KUKA KRL program: ho_st600_r1_1.src, ho_st600_r1_1.dat

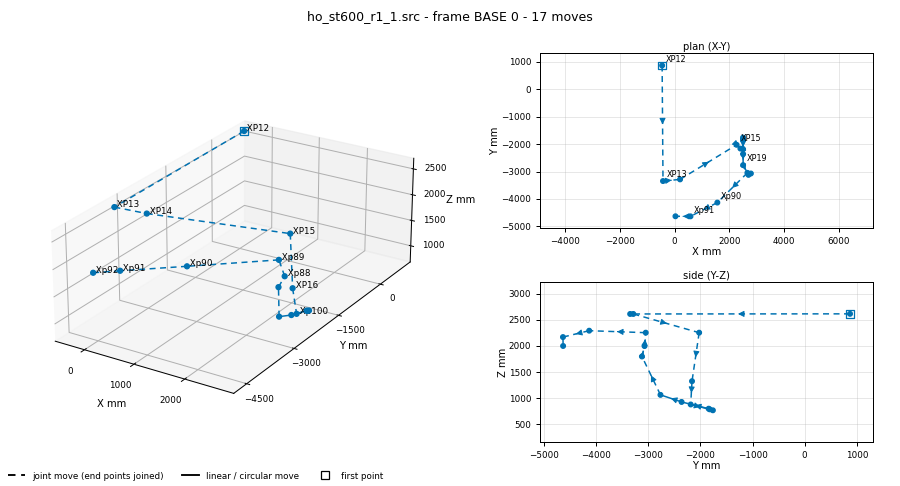
[picture p0: tool path of ho_st600_r1_1.src in frame BASE 0, 17 of 18 moves have a stored position in this frame; points joined in program order, loops and branches not executed]
--- ho_st600_r1_1.src ---
&ACCESS RVO1
&REL 93
&COMMENT Pega traseira ACTROS
&PARAM DISKPATH = KRC:\R1\Program
DEF HO_ST600_R1_1( )
;FOLD INI
  ;FOLD BASISTECH INI
    GLOBAL INTERRUPT DECL 3 WHEN $STOPMESS==TRUE DO IR_STOPM ( )
    INTERRUPT ON 3
    BAS (#INITMOV,0 )
  ;ENDFOLD (BASISTECH INI)
;FOLD GRIPPERTECH INI
USER_GRP(0,DUMMY,DUMMY,GDEFAULT)
;ENDFOLD (GRIPPERTECH INI)
  ;FOLD USER INI
    ;Make your modifications here

  ;ENDFOLD (USER INI)
;ENDFOLD (INI)

; Caracterização dos meios de produção:
; Versão Atual:
; 08/06/2013 12:00 Name: P13.050-R1 CHANGES: Pega Traseira
; Actros MGS\MGSB\LTA\LTB e STB12-13

chk_w5_wechs_ok ( )              ; CHECK GRIPPER ACTROS

;FOLD PTP P12 CONT Vel=100 % PDAT11 Tool[5]:Painel Traseiro Actros Base[0];%{PE}%R 8.2.19,%MKUKATPBASIS,%CMOVE,%VPTP,%P 1:PTP, 2:P12, 3:C_DIS, 5:100, 7:PDAT11
$BWDSTART=FALSE
PDAT_ACT=PPDAT11
FDAT_ACT=FP12
BAS(#PTP_PARAMS,100)
PTP XP12 C_DIS
;ENDFOLD
;FOLD PTP P13 Vel=100 % PDAT12 Tool[5]:Painel Traseiro Actros Base[0];%{PE}%R 8.2.20,%MKUKATPBASIS,%CMOVE,%VPTP,%P 1:PTP, 2:P13, 3:, 5:100, 7:PDAT12
$BWDSTART=FALSE
PDAT_ACT=PPDAT12
FDAT_ACT=FP13
BAS(#PTP_PARAMS,100)
PTP XP13
;ENDFOLD

;FOLD OUT 3352 'R1 busca traseira' State=TRUE ;%{PE}%R 8.2.20,%MKUKATPBASIS,%COUT,%VOUTX,%P 2:3352, 3:R1 busca traseira, 5:TRUE, 6:
$OUT[3352]=TRUE
;ENDFOLD
;FOLD WAIT FOR ( IN 3352 'Aguarda lib. Buscar traseira' );%{PE}%R 8.2.20,%MKUKATPBASIS,%CEXT_WAIT_FOR,%VEXT_WAIT_FOR,%P 2:, 4:, 5:$IN, 6:3352, 7:Aguarda lib. Buscar traseira, 9:
WAIT FOR  ( $IN[3352] )
;ENDFOLD
;FOLD OUT 3352 'R1 busca traseira' State=FALSE ;%{PE}%R 8.2.20,%MKUKATPBASIS,%COUT,%VOUTX,%P 2:3352, 3:R1 busca traseira, 5:FALSE, 6:
$OUT[3352]=FALSE
;ENDFOLD

;FOLD PTP P14 CONT Vel=100 % PDAT13 Tool[5]:Painel Traseiro Actros Base[0];%{PE}%R 8.2.19,%MKUKATPBASIS,%CMOVE,%VPTP,%P 1:PTP, 2:P14, 3:C_DIS, 5:100, 7:PDAT13
$BWDSTART=FALSE
PDAT_ACT=PPDAT13
FDAT_ACT=FP14
BAS(#PTP_PARAMS,100)
PTP XP14 C_DIS
;ENDFOLD
;FOLD PTP P15 CONT Vel=100 % PDAT14 Tool[5]:Painel Traseiro Actros Base[0];%{PE}%R 8.2.19,%MKUKATPBASIS,%CMOVE,%VPTP,%P 1:PTP, 2:P15, 3:C_DIS, 5:100, 7:PDAT14
$BWDSTART=FALSE
PDAT_ACT=PPDAT14
FDAT_ACT=FP15
BAS(#PTP_PARAMS,100)
PTP XP15 C_DIS
;ENDFOLD
;FOLD PTP P16 CONT Vel=100 % PDAT15 Tool[5]:Painel Traseiro Actros Base[0];%{PE}%R 8.2.19,%MKUKATPBASIS,%CMOVE,%VPTP,%P 1:PTP, 2:P16, 3:C_DIS, 5:100, 7:PDAT15
$BWDSTART=FALSE
PDAT_ACT=PPDAT15
FDAT_ACT=FP16
BAS(#PTP_PARAMS,100)
PTP XP16 C_DIS
;ENDFOLD

;FOLD OUT 3342 'Fora area externa' State=FALSE ;%{PE}%R 8.2.20,%MKUKATPBASIS,%COUT,%VOUTX,%P 2:3342, 3:Fora area externa, 5:FALSE, 6:
$OUT[3342]=FALSE
;ENDFOLD

;FOLD SET Z2.1/2 GRP ACTROS State= GDAT2;%{PE}%R 8.2.1,%MKUKATPGRP,%CGRP,%VGRP,%P 2:1, 4:1, 5:#NO, 6:GDAT2, 8:0, 10:0
H50(GRP,1,1,GGDAT2)
;ENDFOLD
chk_w5_grp2_opn()
;FOLD SET Z3.1/2 GRP ACTROS State=OPN GDAT3;%{PE}%R 8.2.1,%MKUKATPGRP,%CGRP,%VGRP,%P 2:2, 4:1, 5:#NO, 6:GDAT3, 8:0, 10:0
H50(GRP,2,1,GGDAT3)
;ENDFOLD
chk_w5_grp3_opn()

;FOLD PTP p100 CONT Vel=100 % PDAT71 Tool[5]:Painel Traseiro Actros Base[0];%{PE}%R 8.2.20,%MKUKATPBASIS,%CMOVE,%VPTP,%P 1:PTP, 2:p100, 3:C_DIS, 5:100, 7:PDAT71
$BWDSTART=FALSE
PDAT_ACT=PPDAT71
FDAT_ACT=Fp100
BAS(#PTP_PARAMS,100)
PTP Xp100 C_DIS
;ENDFOLD
;FOLD PTP p102 CONT Vel=100 % PDAT73 Tool[5]:Painel Traseiro Actros Base[0];%{PE}%R 8.2.20,%MKUKATPBASIS,%CMOVE,%VPTP,%P 1:PTP, 2:p102, 3:C_DIS, 5:100, 7:PDAT73
$BWDSTART=FALSE
PDAT_ACT=PPDAT73
FDAT_ACT=Fp102
BAS(#PTP_PARAMS,100)
PTP Xp102 C_DIS
;ENDFOLD

;FOLD ; POSICAO DE PEGA DA PECA;%{PE}%R 8.2.20,%MKUKATPBASIS,%CCOMMENT,%VNORMAL,%P 2:POSICAO  DE  PEGA  DA  PECA
;ENDFOLD
;FOLD LIN P18 Vel=0.5 m/s CPDAT1 Tool[5]:Painel Traseiro Actros Base[0];%{PE}%R 8.2.20,%MKUKATPBASIS,%CMOVE,%VLIN,%P 1:LIN, 2:P18, 3:, 5:0.5, 7:CPDAT1
$BWDSTART=FALSE
LDAT_ACT=LCPDAT1
FDAT_ACT=FP18
BAS(#CP_PARAMS,0.5)
LIN XP18
;ENDFOLD

IF (NOT(GHOST())) THEN
;FOLD WAIT FOR ( IN 1 'Presença de peça 1 - Actros Todos' ) AND ( IN 2 'Presença de peça 2 - Actros Todos' );%{PE}%R 8.2.20,%MKUKATPBASIS,%CEXT_WAIT_FOR,%VEXT_WAIT_FOR,%P 2:, 4:, 5:$IN, 6:1, 7:Presença de peça 1 - Actros Todos, 9:AND, 10:, 12:, 13:$IN, 14:2, 15:Presença de peça 2 - Actros Todos, 17:
WAIT FOR  ( $IN[1] ) AND ( $IN[2] )
;ENDFOLD
ENDIF

;FOLD SET Z2.1/2 GRP ACTROS State=CLO GDAT1;%{PE}%R 8.2.1,%MKUKATPGRP,%CGRP,%VGRP,%P 2:1, 4:2, 5:#NO, 6:GDAT1, 8:0, 10:0
H50(GRP,1,2,GGDAT1)
;ENDFOLD
chk_w5_grp2_clo()
;FOLD SET Z3.1/2 GRP ACTROS State=CLO GDAT4;%{PE}%R 8.2.1,%MKUKATPGRP,%CGRP,%VGRP,%P 2:2, 4:2, 5:#NO, 6:GDAT4, 8:0, 10:0
H50(GRP,2,2,GGDAT4)
;ENDFOLD
chk_w5_grp3_clo()

IF (NOT(GHOST())) THEN
;FOLD SET Ventosa ACTROS State=VACUUM GDAT5;%{PE}%R 8.2.1,%MKUKATPGRP,%CGRP,%VGRP,%P 2:6, 4:1, 5:#NO, 6:GDAT5, 8:0, 10:0
H50(GRP,6,1,GGDAT5)
;ENDFOLD
;chk_w5_grp1_vac()
ENDIF

;FOLD OUT 3350 'Solicita lib sair magazine' State=TRUE ;%{PE}%R 8.2.20,%MKUKATPBASIS,%COUT,%VOUTX,%P 2:3350, 3:Solicita lib sair magazine, 5:TRUE, 6:
$OUT[3350]=TRUE
;ENDFOLD
;FOLD WAIT FOR ( IN 3349 'Aguarda lib sair magazine' );%{PE}%R 8.2.20,%MKUKATPBASIS,%CEXT_WAIT_FOR,%VEXT_WAIT_FOR,%P 2:, 4:, 5:$IN, 6:3349, 7:Aguarda lib sair magazine, 9:
WAIT FOR  ( $IN[3349] )
;ENDFOLD
;FOLD OUT 3350 'Solicita lib sair magazine' State=FALSE ;%{PE}%R 8.2.20,%MKUKATPBASIS,%COUT,%VOUTX,%P 2:3350, 3:Solicita lib sair magazine, 5:FALSE, 6:
$OUT[3350]=FALSE
;ENDFOLD
;FOLD OUT 3349 'R1 Pegou peca' State=FALSE ;%{PE}%R 8.2.20,%MKUKATPBASIS,%COUT,%VOUTX,%P 2:3349, 3:R1 Pegou peca, 5:FALSE, 6:
$OUT[3349]=FALSE
;ENDFOLD

;FOLD LIN p101 CONT Vel=1 m/s CPDAT12 Tool[5]:Painel Traseiro Actros Base[0];%{PE}%R 8.2.20,%MKUKATPBASIS,%CMOVE,%VLIN,%P 1:LIN, 2:p101, 3:C_DIS C_DIS, 5:1, 7:CPDAT12
$BWDSTART=FALSE
LDAT_ACT=LCPDAT12
FDAT_ACT=Fp101
BAS(#CP_PARAMS,1)
LIN Xp101 C_DIS C_DIS
;ENDFOLD
;FOLD LIN p95 CONT Vel=1 m/s CPDAT11 Tool[5]:Painel Traseiro Actros Base[0];%{PE}%R 8.2.20,%MKUKATPBASIS,%CMOVE,%VLIN,%P 1:LIN, 2:p95, 3:C_DIS C_DIS, 5:1, 7:CPDAT11
$BWDSTART=FALSE
LDAT_ACT=LCPDAT11
FDAT_ACT=Fp95
BAS(#CP_PARAMS,1)
LIN Xp95 C_DIS C_DIS
;ENDFOLD

IF (NOT(GHOST())) THEN
;FOLD WAIT FOR ( IN 1 'Presença de peça 1 - Actros Todos' ) AND ( IN 2 'Presença de peça 2 - Actros Todos' );%{PE}%R 8.2.20,%MKUKATPBASIS,%CEXT_WAIT_FOR,%VEXT_WAIT_FOR,%P 2:, 4:, 5:$IN, 6:1, 7:Presença de peça 1 - Actros Todos, 9:AND, 10:, 12:, 13:$IN, 14:2, 15:Presença de peça 2 - Actros Todos, 17:
WAIT FOR  ( $IN[1] ) AND ( $IN[2] )
;ENDFOLD
ENDIF

;FOLD LIN P19 Vel=1.5 m/s CPDAT2 Tool[5]:Painel Traseiro Actros Base[0];%{PE}%R 8.2.20,%MKUKATPBASIS,%CMOVE,%VLIN,%P 1:LIN, 2:P19, 3:, 5:1.5, 7:CPDAT2
$BWDSTART=FALSE
LDAT_ACT=LCPDAT2
FDAT_ACT=FP19
BAS(#CP_PARAMS,1.5)
LIN XP19
;ENDFOLD

;FOLD PTP P21 CONT Vel=100 % PDAT19 Tool[5]:Painel Traseiro Actros Base[0];%{PE}%R 8.2.19,%MKUKATPBASIS,%CMOVE,%VPTP,%P 1:PTP, 2:P21, 3:C_DIS, 5:100, 7:PDAT19
$BWDSTART=FALSE
PDAT_ACT=PPDAT19
FDAT_ACT=FP21
BAS(#PTP_PARAMS,100)
PTP XP21 C_DIS
;ENDFOLD
;FOLD PTP p88 CONT Vel=100 % PDAT60 Tool[5]:Painel Traseiro Actros Base[0];%{PE}%R 8.2.19,%MKUKATPBASIS,%CMOVE,%VPTP,%P 1:PTP, 2:p88, 3:C_DIS, 5:100, 7:PDAT60
$BWDSTART=FALSE
PDAT_ACT=PPDAT60
FDAT_ACT=Fp88
BAS(#PTP_PARAMS,100)
PTP Xp88 C_DIS
;ENDFOLD
;FOLD PTP p89 CONT Vel=100 % PDAT61 Tool[5]:Painel Traseiro Actros Base[0];%{PE}%R 8.2.19,%MKUKATPBASIS,%CMOVE,%VPTP,%P 1:PTP, 2:p89, 3:C_DIS, 5:100, 7:PDAT61
$BWDSTART=FALSE
PDAT_ACT=PPDAT61
FDAT_ACT=Fp89
BAS(#PTP_PARAMS,100)
PTP Xp89 C_DIS
;ENDFOLD
;FOLD PTP p90 CONT Vel=80 % PDAT62 Tool[5]:Painel Traseiro Actros Base[0];%{PE}%R 8.2.19,%MKUKATPBASIS,%CMOVE,%VPTP,%P 1:PTP, 2:p90, 3:C_DIS, 5:80, 7:PDAT62
$BWDSTART=FALSE
PDAT_ACT=PPDAT62
FDAT_ACT=Fp90
BAS(#PTP_PARAMS,80)
PTP Xp90 C_DIS
;ENDFOLD
;FOLD PTP p91 CONT Vel=80 % PDAT63 Tool[5]:Painel Traseiro Actros Base[0];%{PE}%R 8.2.19,%MKUKATPBASIS,%CMOVE,%VPTP,%P 1:PTP, 2:p91, 3:C_DIS, 5:80, 7:PDAT63
$BWDSTART=FALSE
PDAT_ACT=PPDAT63
FDAT_ACT=Fp91
BAS(#PTP_PARAMS,80)
PTP Xp91 C_DIS
;ENDFOLD

;FOLD PTP p92 CONT Vel=80 % PDAT64 Tool[5]:Painel Traseiro Actros Base[0];%{PE}%R 8.2.19,%MKUKATPBASIS,%CMOVE,%VPTP,%P 1:PTP, 2:p92, 3:C_DIS, 5:80, 7:PDAT64
$BWDSTART=FALSE
PDAT_ACT=PPDAT64
FDAT_ACT=Fp92
BAS(#PTP_PARAMS,80)
PTP Xp92 C_DIS
;ENDFOLD

;FOLD Collision.Monitoring_AREA_5_On ;%{PE}%MKUKATPUSER
COLLSTOP( 11, 1 ) ;not Interrupt-Controlled
;ENDFOLD

;FOLD PTP HOME3 Vel=100 % PDAT59;%{PE}%R 8.2.19,%MKUKATPBASIS,%CMOVE,%VPTP,%P 1:PTP, 2:HOME3, 3:, 5:100, 7:PDAT59
$BWDSTART=FALSE
PDAT_ACT=PPDAT59
FDAT_ACT=FHOME3
BAS(#PTP_PARAMS,100)
PTP XHOME3
;ENDFOLD

;FOLD OUT 3349 'R1 Pegou peca' State=TRUE ;%{PE}%R 8.2.20,%MKUKATPBASIS,%COUT,%VOUTX,%P 2:3349, 3:R1 Pegou peca, 5:TRUE, 6:
$OUT[3349]=TRUE
;ENDFOLD
;FOLD OUT 3342 'Fora area externa' State=TRUE ;%{PE}%R 8.2.20,%MKUKATPBASIS,%COUT,%VOUTX,%P 2:3342, 3:Fora area externa, 5:TRUE, 6:
$OUT[3342]=TRUE
;ENDFOLD

END

--- ho_st600_r1_1.dat ---
&ACCESS RVO1
&REL 93
&COMMENT Pega traseira ACTROS
&PARAM DISKPATH = KRC:\R1\Program
DEFDAT  HO_ST600_R1_1
;FOLD EXTERNAL DECLARATIONS;%{PE}%MKUKATPBASIS,%CEXT,%VCOMMON,%P
;FOLD GRIPPERTECH EXT
EXT  H50 (INT  :IN,INT  :IN,INT  :IN,GRP_TYP  :IN )
;ENDFOLD (GRIPPERTECH EXT)
;FOLD SPOTTECH EXT
EXT  USERSPOT (S_COMMAND  :IN,SPOT_TYPE  :IN )
;ENDFOLD (SPOTTECH EXT)
;FOLD BASISTECH EXT;%{PE}%MKUKATPBASIS,%CEXT,%VEXT,%P
EXT  BAS (BAS_COMMAND  :IN,REAL  :IN )
DECL INT SUCCESS
;ENDFOLD (BASISTECH EXT)
;FOLD USER EXT;%{E}%MKUKATPUSER,%CEXT,%VEXT,%P
;Make your modifications here

;ENDFOLD (USER EXT)
;ENDFOLD (EXTERNAL DECLARATIONS)

;# ============ START PATH : bh_p13050r1_lta_01 =============
DECL BASIS_SUGG_T LAST_BASIS={POINT1[] "p102                    ",POINT2[] "p102                    ",CP_PARAMS[] "CPDAT11                 ",PTP_PARAMS[] "PDAT73                  ",CONT[] "C_DIS                   ",CP_VEL[] "1.5                     ",PTP_VEL[] "100                     ",SYNC_PARAMS[] "SYNCDAT                 ",SPL_NAME[] "S0                      "}
DECL PDAT PPDAT11={VEL 100.0,ACC 100.0,APO_DIST 100.0,APO_MODE #CDIS}
DECL E6POS XP12={X -451.816589,Y 870.27887,Z 2616.43896,A -71.9595718,B 86.8192902,C 144.022598,S 2,T 11,E1 -267.097687,E2 0.0,E3 0.0,E4 0.0,E5 0.0,E6 0.0}
DECL FDAT FP12={TOOL_NO 5,BASE_NO 0,IPO_FRAME #BASE,POINT2[] " ",TQ_STATE FALSE}
DECL PDAT PPDAT12={VEL 100.0,ACC 100.0,APO_DIST 100.0,APO_MODE #CDIS}
DECL E6POS XP13={X -419.798889,Y -3347.46606,Z 2614.177,A -64.8434372,B 86.6851501,C 143.229507,S 2,T 11,E1 -4438.06104,E2 0.0,E3 0.0,E4 0.0,E5 0.0,E6 0.0}
DECL FDAT FP13={TOOL_NO 5,BASE_NO 0,IPO_FRAME #BASE,POINT2[] " ",TQ_STATE FALSE}
DECL PDAT PPDAT13={VEL 100.0,ACC 100.0,APO_DIST 100.0,APO_MODE #CDIS}
DECL E6POS XP14={X 202.780197,Y -3287.19092,Z 2614.17407,A -95.8952332,B 86.6846771,C 143.223602,S 2,T 11,E1 -4438.06104,E2 0.0,E3 0.0,E4 0.0,E5 0.0,E6 0.0}
DECL FDAT FP14={TOOL_NO 5,BASE_NO 0,IPO_FRAME #BASE,POINT2[] " ",TQ_STATE FALSE}
DECL PDAT PPDAT14={VEL 100.0,ACC 100.0,APO_DIST 100.0,APO_MODE #CDIS}
DECL E6POS XP15={X 2268.02295,Y -2024.03894,Z 2255.53906,A -43.859211,B 87.126442,C -132.618103,S 2,T 11,E1 -3004.49902,E2 0.0,E3 0.0,E4 0.0,E5 0.0,E6 0.0}
DECL FDAT FP15={TOOL_NO 5,BASE_NO 0,IPO_FRAME #BASE,POINT2[] " ",TQ_STATE FALSE}
DECL PDAT PPDAT15={VEL 100.0,ACC 100.0,APO_DIST 100.0,APO_MODE #CDIS}
DECL E6POS XP16={X 2406.44995,Y -2161.04907,Z 1324.771,A -90.5126572,B 68.1089096,C -177.290695,S 2,T 11,E1 -2729.26611,E2 0.0,E3 0.0,E4 0.0,E5 0.0,E6 0.0}
DECL FDAT FP16={TOOL_NO 5,BASE_NO 0,IPO_FRAME #BASE,POINT2[] " ",TQ_STATE FALSE}
DECL LDAT LCPDAT1={VEL 2.0,ACC 100.0,APO_DIST 100.0,APO_FAC 50.0,AXIS_VEL 100.0,AXIS_ACC 100.0,ORI_TYP #VAR,CIRC_TYP #BASE,JERK_FAC 50.0,GEAR_JERK 50.0,EXAX_IGN 0}
DECL E6POS XP18={X 2502.87012,Y -1760.80396,Z 766.271484,A -89.9168472,B 75.7216568,C -179.767197,S 2,T 11,E1 -2729.85596,E2 0.0,E3 0.0,E4 0.0,E5 0.0,E6 0.0}
DECL FDAT FP18={TOOL_NO 5,BASE_NO 0,IPO_FRAME #BASE,POINT2[] " ",TQ_STATE FALSE}
DECL E6POS XP19={X 2504.81006,Y -2766.26196,Z 1062.104,A -90.0798721,B 75.6205063,C -179.986496,S 2,T 11,E1 -2985.20703,E2 0.0,E3 0.0,E4 0.0,E5 0.0,E6 0.0}
DECL FDAT FP19={TOOL_NO 5,BASE_NO 0,IPO_FRAME #BASE,POINT2[] " ",TQ_STATE FALSE}
DECL LDAT LCPDAT2={VEL 2.0,ACC 100.0,APO_DIST 100.0,APO_FAC 50.0,AXIS_VEL 100.0,AXIS_ACC 100.0,ORI_TYP #VAR,CIRC_TYP #BASE,JERK_FAC 50.0,GEAR_JERK 50.0,EXAX_IGN 0}
DECL E6POS XP21={X 2700.63306,Y -3121.27197,Z 1798.22095,A -162.698898,B 78.5070572,C 171.130295,S 2,T 11,E1 -3279.66504,E2 0.0,E3 0.0,E4 0.0,E5 0.0,E6 0.0}
DECL FDAT FP21={TOOL_NO 5,BASE_NO 0,IPO_FRAME #BASE,POINT2[] " ",TQ_STATE FALSE}
DECL PDAT PPDAT19={VEL 100.0,ACC 100.0,APO_DIST 100.0,APO_MODE #CDIS}
DECL FDAT FHOME3={TOOL_NO 5,BASE_NO 0,IPO_FRAME #BASE,POINT2[] " ",TQ_STATE FALSE}
DECL PDAT PPDAT59={VEL 100.0,ACC 100.0,APO_DIST 100.0,APO_MODE #CDIS}
DECL E6POS XP88={X 2788.45605,Y -3071.81201,Z 1998.68799,A -179.131805,B 83.0067825,C -178.304398,S 6,T 27,E1 -2884.48804,E2 0.0,E3 0.0,E4 0.0,E5 0.0,E6 0.0}
DECL FDAT Fp88={TOOL_NO 5,BASE_NO 0,IPO_FRAME #BASE,POINT2[] " ",TQ_STATE FALSE}
DECL PDAT PPDAT60={VEL 100.0,ACC 100.0,APO_DIST 100.0,APO_MODE #CDIS}
DECL PDAT PPDAT61={VEL 100.0,ACC 100.0,APO_DIST 100.0,APO_MODE #CDIS}
DECL E6POS Xp89={X 2660.87988,Y -3048.35303,Z 2255.20996,A -123.1717,B 88.586731,C -92.6604538,S 6,T 27,E1 -2443.08496,E2 0.0,E3 0.0,E4 0.0,E5 0.0,E6 0.0}
DECL FDAT Fp89={TOOL_NO 5,BASE_NO 0,IPO_FRAME #BASE,POINT2[] " ",TQ_STATE FALSE}
DECL PDAT PPDAT62={VEL 100.0,ACC 100.0,APO_DIST 100.0,APO_MODE #CDIS}
DECL E6POS Xp90={X 1564.13794,Y -4133.34912,Z 2293.29907,A -41.9511108,B 87.0503387,C 35.2014198,S 6,T 27,E1 -2224.604,E2 0.0,E3 0.0,E4 0.0,E5 0.0,E6 0.0}
DECL FDAT Fp90={TOOL_NO 5,BASE_NO 0,IPO_FRAME #BASE,POINT2[] " ",TQ_STATE FALSE}
DECL PDAT PPDAT63={VEL 100.0,ACC 100.0,APO_DIST 100.0,APO_MODE #CDIS}
DECL E6POS Xp91={X 583.737183,Y -4636.52197,Z 2170.92603,A -1.58821595,B 78.5376968,C 92.3479614,S 6,T 26,E1 -2650.03394,E2 0.0,E3 0.0,E4 0.0,E5 0.0,E6 0.0}
DECL FDAT Fp91={TOOL_NO 5,BASE_NO 0,IPO_FRAME #BASE,POINT2[] " ",TQ_STATE FALSE}
DECL PDAT PPDAT64={VEL 100.0,ACC 100.0,APO_DIST 100.0,APO_MODE #CDIS}
DECL E6POS Xp92={X 34.7994919,Y -4633.68994,Z 2000.20996,A -0.689865112,B 78.3299789,C 94.622963,S 6,T 26,E1 -2650.04102,E2 0.0,E3 0.0,E4 0.0,E5 0.0,E6 0.0}
DECL FDAT Fp92={TOOL_NO 5,BASE_NO 0,IPO_FRAME #BASE,POINT2[] " ",TQ_STATE FALSE}
DECL E6POS XP95={X 2505.06396,Y -2361.08496,Z 926.497681,A -90.0794373,B 75.6205673,C -179.985901,S 2,T 11,E1 -2729.68311,E2 0.0,E3 0.0,E4 0.0,E5 0.0,E6 0.0}
DECL FDAT Fp95={TOOL_NO 5,BASE_NO 0,IPO_FRAME #BASE,POINT2[] " ",TQ_STATE FALSE}
DECL LDAT LCPDAT11={VEL 2.0,ACC 100.0,APO_DIST 100.0,APO_FAC 50.0,AXIS_VEL 100.0,AXIS_ACC 100.0,ORI_TYP #VAR,CIRC_TYP #BASE,JERK_FAC 50.0,GEAR_JERK 50.0,EXAX_IGN 0}
DECL GRP_SUGG_T LAST_GRP={NUMBER[] "6                       ",STATE[] "1                       ",PARAMS[] "GDAT5                   "}
DECL GRP_TYP GGDAT1={G_APO #NO,GRP_TIME 0.200000003,CTRL #OFF,DLY 0,DST 1}
DECL GRP_TYP GGDAT2={G_APO #NO,GRP_TIME 0.200000003,CTRL #OFF,DLY 0,DST 1}
DECL GRP_TYP GGDAT3={G_APO #NO,GRP_TIME 0.200000003,CTRL #OFF,DLY 0,DST 1}
DECL GRP_TYP GGDAT4={G_APO #NO,GRP_TIME 0.200000003,CTRL #OFF,DLY 0,DST 1}
DECL PDAT PPDAT71={VEL 100.0,ACC 100.0,APO_DIST 100.0,APO_MODE #CDIS}
DECL E6POS Xp100={X 2505.35205,Y -2186.28198,Z 877.875305,A -90.0798569,B 75.6182938,C -179.986099,S 2,T 11,E1 -2729.66699,E2 0.0,E3 0.0,E4 0.0,E5 0.0,E6 0.0}
DECL FDAT Fp100={TOOL_NO 5,BASE_NO 0,IPO_FRAME #BASE,POINT2[] " ",TQ_STATE FALSE}
DECL GRP_TYP GGDAT5={G_APO #NO,GRP_TIME 0.200000003,CTRL #OFF,DLY 0,DST 1}
DECL E6POS XP101={X 2503.15991,Y -1841.73206,Z 797.207581,A -89.4281387,B 75.7452011,C -179.251404,S 2,T 11,E1 -2729.66406,E2 0.0,E3 0.0,E4 0.0,E5 0.0,E6 0.0}
DECL FDAT Fp101={TOOL_NO 5,BASE_NO 0,IPO_FRAME #BASE,POINT2[] " ",TQ_STATE FALSE}
DECL LDAT LCPDAT12={VEL 2.0,ACC 100.0,APO_DIST 100.0,APO_FAC 50.0,AXIS_VEL 100.0,AXIS_ACC 100.0,ORI_TYP #VAR,CIRC_TYP #BASE,JERK_FAC 50.0,GEAR_JERK 50.0,EXAX_IGN 0}
DECL E6POS XP102={X 2504.4751,Y -1821.45203,Z 784.470825,A -90.2340164,B 75.7273331,C 179.802094,S 2,T 11,E1 -2729.87305,E2 0.0,E3 0.0,E4 0.0,E5 0.0,E6 0.0}
DECL FDAT Fp102={TOOL_NO 5,BASE_NO 0,IPO_FRAME #BASE,POINT2[] " ",TQ_STATE FALSE}
DECL PDAT PPDAT73={VEL 100.0,ACC 100.0,APO_DIST 100.0,APO_MODE #CDIS}
ENDDAT
